FUNCTION FinishAction 
VAR_INPUT
	StartAsync : BOOL := FALSE;
	StopAsync : BOOL :=FALSE;
END_VAR
VAR
END_VAR

IF StopAsync THEN 
	G_Match.iAsyncAction := ''; 
	G_Match.iEtapeAction := 0;
ELSE
	G_Match.bActionFinie := TRUE;
	IF NOT StartAsync THEN 
		G_Match.iAsyncAction := ''; 
		G_Match.iEtapeAction := 0;
	END_IF
END_IF

END_FUNCTION

(* stored: Version 1.1.0.1, ProductVersion 3.1.4024.11
   POU FinishAction: Id {64a2e075-7474-4a98-af0d-323ec0420576}, SpecialFunc None *)
